// TIA Portal V19 export
FUNCTION_BLOCK "CallGlobal"   // FB48, LAD
TITLE = CallGlobal
// All blocks that provide data to the DB Global.Data are called here. That includes blocks to generate system data as well as blocks that connect handle multiple HMIs.
// stored: IsIECCheckEnabled true, MemoryReserve 100, SetENOAutomatically true
   VAR
      statClockSysMemOld { ExternalWritable := 'False'} : Byte;   // Old value system memory evaluation / Alter Wert Systeminformationsspeicher auswertung
      instLAF_PowerOnOff { ExternalWritable := 'False'} : "LAF_PowerOnOff";
      instLAF_HmiHeaderManager { ExternalWritable := 'False'} : "LAF_HmiHeaderManager";
      instLAF_ClockGen { ExternalWritable := 'False'} : "LAF_ClockGenerator";
      instLSNTP_Server { ExternalWritable := 'False'} : "LSNTP_Server";
   END_VAR
   VAR_TEMP
      tempIndex : DInt;   // Temp variable for for loop
      tempAcknowledge : Bool;   // Summarized acknowledge command
      tempPowerOff : Bool;   // Summarized power off command
      tempPowerOn : Bool;   // Summarized power on command
      tempPowerStatus : Int;   // 0 - Off, 1 - Paused, 2 - On
      tempResultXor : Byte;   // Interim result of XOR operation / Zwischenergebnis von XOR Anweisung
      tempPosPulse : Byte;   // Interim result puls calculation / Zwischenergebnis von Pulsauswertung
   END_VAR
   VAR CONSTANT
      RESET_BUTTON__COULD_BE_ADDED_HERE : Bool := false;   // Placeholder for a potential global reset button
   END_VAR
BEGIN

REGION Network 1 (SCL): Summarize HMI commands
   // Read commands for acknowledge, powerOn and powerOff from the different HMI panels and summarize them in temp variables for further logic in this block.
   // Initialize temp variables
   #tempAcknowledge :=
   #tempPowerOff :=
   #tempPowerOn := FALSE;

   // Loop through the HMI panels and summarize the commands
   FOR #tempIndex := 0 TO "NO_OF_PANELS" DO
       #tempAcknowledge := #tempAcknowledge OR "Hmi".mainHeader[#tempIndex].hmiToPlc.acknowledge;
       #tempPowerOff := #tempPowerOff OR "Hmi".mainHeader[#tempIndex].hmiToPlc.powerCommands.%X0;
       #tempPowerOn := #tempPowerOn OR "Hmi".mainHeader[#tempIndex].hmiToPlc.powerCommands.%X1;
   END_FOR;
END_REGION

REGION Network 2: Global Acknowledge
   // The global acknowledge command from the hmi button is assigned to Global.Data.general.acknowledge: This bit it forwarded to all underlaying modules
   // If a hard-wired global reset button exists, it can
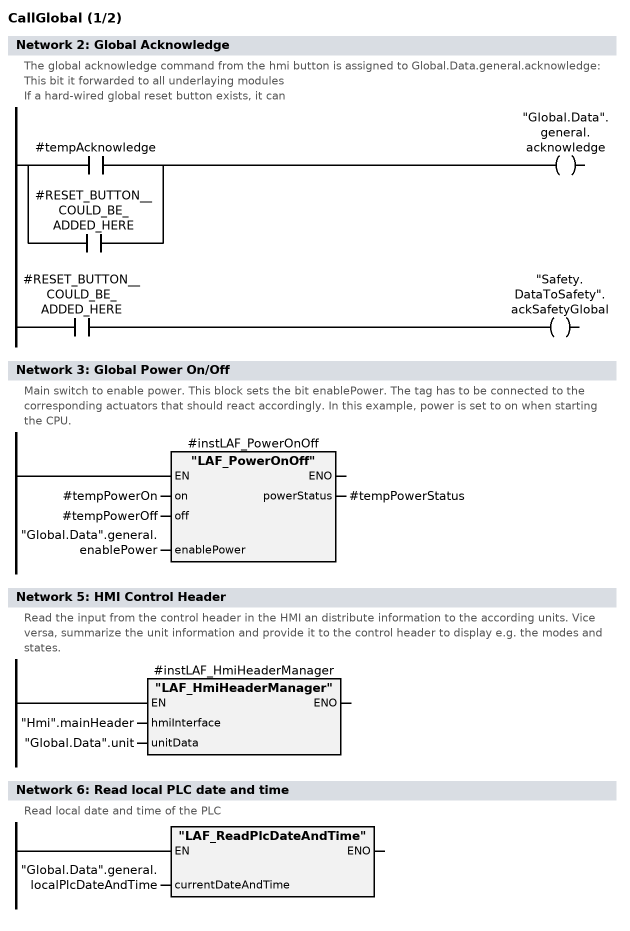
   RUNG wire#powerrail
      Contact( #tempAcknowledge )
      wire#w1
      Coil( "Global.Data".general.acknowledge )
   END_RUNG
   RUNG wire#powerrail
      Contact( #RESET_BUTTON__COULD_BE_ADDED_HERE )
   END_RUNG wire#w1
   RUNG wire#powerrail
      Contact( #RESET_BUTTON__COULD_BE_ADDED_HERE )
      Coil( "Safety.DataToSafety".ackSafetyGlobal )
   END_RUNG
   // the same network as SCL:
   "Global.Data".general.acknowledge := #tempAcknowledge OR #RESET_BUTTON__COULD_BE_ADDED_HERE;
   "Safety.DataToSafety".ackSafetyGlobal := #RESET_BUTTON__COULD_BE_ADDED_HERE;
END_REGION

REGION Network 3: Global Power On/Off
   // Main switch to enable power. This block sets the bit enablePower. The tag has to be connected to the corresponding actuators that should react accordingly. In this example, power is set to on when starting the CPU.
   RUNG wire#powerrail
      #instLAF_PowerOnOff(on := #tempPowerOn, off := #tempPowerOff, enablePower := "Global.Data".general.enablePower, powerStatus => #tempPowerStatus)
   END_RUNG
   // the same network as SCL:
   #instLAF_PowerOnOff(on := #tempPowerOn,   // "LAF_PowerOnOff"
                       off := #tempPowerOff,
                       enablePower := "Global.Data".general.enablePower,
                       powerStatus => #tempPowerStatus);
END_REGION

REGION Network 4 (SCL): Write power status to HMI panels
   // Write power status back to all connected HMI panels
   // Loop through the panels and set the power status
   FOR #tempIndex := 0 TO "NO_OF_PANELS" DO
       "Hmi".mainHeader[#tempIndex].plcToHmi.powerStatus := #tempPowerStatus;
   END_FOR;
END_REGION

REGION Network 5: HMI Control Header
   // Read the input from the control header in the HMI an distribute information to the according units. Vice versa, summarize the unit information and provide it to the control header to display e.g. the modes and states.
   RUNG wire#powerrail
      #instLAF_HmiHeaderManager(hmiInterface := "Hmi".mainHeader, unitData := "Global.Data".unit)
   END_RUNG
   // the same network as SCL:
   #instLAF_HmiHeaderManager(hmiInterface := "Hmi".mainHeader, unitData := "Global.Data".unit);   // "LAF_HmiHeaderManager"
END_REGION

REGION Network 6: Read local PLC date and time
   // Read local date and time of the PLC
   RUNG wire#powerrail
      "LAF_ReadPlcDateAndTime"(currentDateAndTime := "Global.Data".general.localPlcDateAndTime)
   END_RUNG
   // the same network as SCL:
   "LAF_ReadPlcDateAndTime"(currentDateAndTime := "Global.Data".general.localPlcDateAndTime);
END_REGION

REGION Network 7: Create clock bits / Takt Bits erstellen
   // The clock bits are generated instead of the HW clock memory byte of the PLC. Due to the use of software units, the ussage of system and clock memory bytes isn't possible. / Die Taktbits werden erzeugt anstelle der HW Taktmerker Byte der SPS. Durch die verwendung von Softwareunits ist der Zugriff auf die System und Taktmerker nicht möglich.
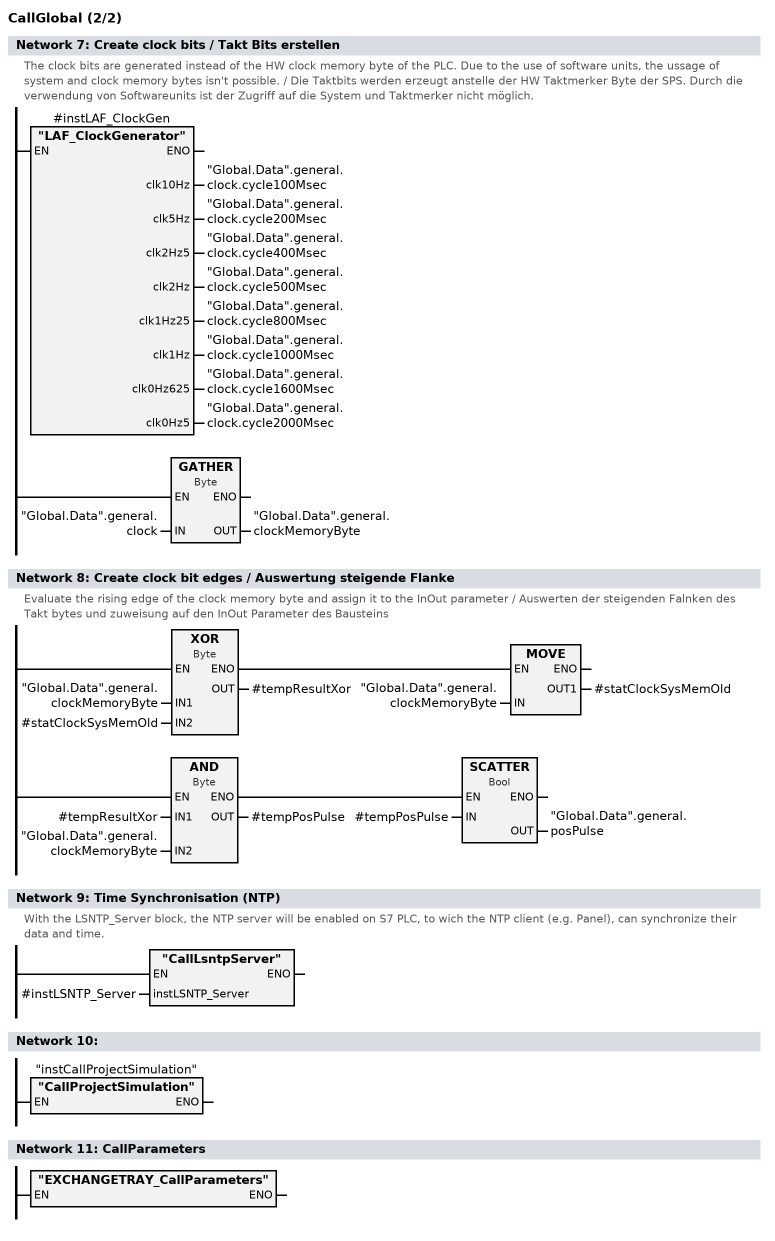
   RUNG wire#powerrail
      #instLAF_ClockGen(clk10Hz => "Global.Data".general.clock.cycle100Msec, clk5Hz => "Global.Data".general.clock.cycle200Msec, clk2Hz5 => "Global.Data".general.clock.cycle400Msec, clk2Hz => "Global.Data".general.clock.cycle500Msec, clk1Hz25 => "Global.Data".general.clock.cycle800Msec, clk1Hz => "Global.Data".general.clock.cycle1000Msec, clk0Hz625 => "Global.Data".general.clock.cycle1600Msec, clk0Hz5 => "Global.Data".general.clock.cycle2000Msec)
   END_RUNG
   RUNG wire#powerrail
      { S7_Templates := "[dest_type := Byte, src_type := Bool]" } GATHER(IN := "Global.Data".general.clock, OUT => "Global.Data".general.clockMemoryByte)
   END_RUNG
   // the same network as SCL:
   #instLAF_ClockGen(clk10Hz => "Global.Data".general.clock.cycle100Msec,   // "LAF_ClockGenerator"
                     clk5Hz => "Global.Data".general.clock.cycle200Msec,
                     clk2Hz5 => "Global.Data".general.clock.cycle400Msec,
                     clk2Hz => "Global.Data".general.clock.cycle500Msec,
                     clk1Hz25 => "Global.Data".general.clock.cycle800Msec,
                     clk1Hz => "Global.Data".general.clock.cycle1000Msec,
                     clk0Hz625 => "Global.Data".general.clock.cycle1600Msec,
                     clk0Hz5 => "Global.Data".general.clock.cycle2000Msec);
   GATHER(IN := "Global.Data".general.clock, OUT => "Global.Data".general.clockMemoryByte);
END_REGION

REGION Network 8: Create clock bit edges / Auswertung steigende Flanke
   // Evaluate the rising edge of the clock memory byte and assign it to the InOut parameter / Auswerten der steigenden Falnken des Takt bytes und zuweisung auf den InOut Parameter des Bausteins
   #tempResultXor := "Global.Data".general.clockMemoryByte XOR #statClockSysMemOld;
   #statClockSysMemOld := "Global.Data".general.clockMemoryByte;
   #tempPosPulse := #tempResultXor AND "Global.Data".general.clockMemoryByte;
   SCATTER(IN := #tempPosPulse, OUT => "Global.Data".general.posPulse);
END_REGION

REGION Network 9: Time Synchronisation (NTP)
   // With the LSNTP_Server block, the NTP server will be enabled on S7 PLC, to wich the NTP client (e.g. Panel), can synchronize their data and time.
   RUNG wire#powerrail
      "CallLsntpServer"(instLSNTP_Server := #instLSNTP_Server)
   END_RUNG
   // the same network as SCL:
   "CallLsntpServer"(instLSNTP_Server := #instLSNTP_Server);
END_REGION

REGION Network 10
   RUNG wire#powerrail
      "instCallProjectSimulation"()
   END_RUNG
   // the same network as SCL:
   "instCallProjectSimulation"();   // "CallProjectSimulation"
END_REGION

REGION Network 11: CallParameters
   RUNG wire#powerrail
      "EXCHANGETRAY_CallParameters"()
   END_RUNG
   // the same network as SCL:
   "EXCHANGETRAY_CallParameters"();
END_REGION
END_FUNCTION_BLOCK
